# EPICS substitutions: db/Beckhoff_7XXX/ecmcEL7332.substitutions
file "ecmcEcSlave.template"
{
  pattern {}
          {}
}

# All fields related to velocity scaling and alarms
file "ecmcEL7332-chX.template"
{
  pattern {CH_ID}
          {01   }
          {02   }
}
